TEXTLIST M2ConfigTabsTextList
  0 = 'General'
  1 = 'X axis'
  2 = 'Y axis'
  3 = 'Z axis (general)'
  4 = 'Z axis (specific)'
  5 = 'Tilt X axis'
  6 = 'Tilt Y axis'
  7 = 'Thermal focus'
   = ''
END_TEXTLIST

(* stored: Version 1.1.0.1, ProductVersion 3.1.4018.5
   TextList M2ConfigTabsTextList: Id {595e8ac0-eff3-422d-bfde-137adcab9bb5} *)
